PROGRAM AdsTcpUnit
VAR_OUTPUT
	bBusy : BOOL;
	err : BOOL;
	errid : UDINT;
END_VAR
VAR_OUTPUT
	areaSockets : ARRAY[1..6] OF POINTER TO AdsSocket; //only used for finding a socket by name
	subarea4Sockets : ARRAY[1..9] OF POINTER TO AdsSocket;
END_VAR
VAR	
	socket : REFERENCE TO AdsSocket;
	i : INT;
END_VAR

(*
this basic version of AdsTcp communication does not dynamically generate ADS messages into a queue to be polled cyclically
instead, modules must wait for the requested socket to finish sending its previous data before sending the next
*)

areaSockets[1] := ADR(AREA_1);
areaSockets[2] := ADR(AREA_2);
areaSockets[3] := ADR(AREA_3);
areaSockets[4] := ADR(AREA_4);
areaSockets[5] := ADR(AREA_5);
areaSockets[6] := ADR(AREA_6);

subarea4Sockets[1] := ADR(SUBAREA_4_1);
subarea4Sockets[2] := ADR(SUBAREA_4_2);
subarea4Sockets[3] := ADR(SUBAREA_4_3);
subarea4Sockets[4] := ADR(SUBAREA_4_4);
subarea4Sockets[5] := ADR(SUBAREA_4_5);
subarea4Sockets[6] := ADR(SUBAREA_4_6);
subarea4Sockets[7] := ADR(SUBAREA_4_7);
subarea4Sockets[8] := ADR(SUBAREA_4_8);
subarea4Sockets[9] := ADR(SUBAREA_4_9);

blocks();

METHOD PRIVATE blocks : BOOL
VAR_INPUT
END_VAR
(*
AREA_1(
	PrgName=> , 
	AmsNetId=> , 
	AmsPort=> , 
	receivingData=> , 
	sendingData=> , 
	readBusy=> , 
	readError=> , 
	readErrorId=> , 
	writeBusy=> , 
	writeError=> , 
	writeErrorId=> );
*)
(*
AREA_2(
	PrgName=> , 
	AmsNetId=> , 
	AmsPort=> , 
	receivingData=> , 
	sendingData=> , 
	readBusy=> , 
	readError=> , 
	readErrorId=> , 
	writeBusy=> , 
	writeError=> , 
	writeErrorId=> );
*)
(*
AREA_3(
	PrgName=> , 
	AmsNetId=> , 
	AmsPort=> , 
	receivingData=> , 
	sendingData=> , 
	readBusy=> , 
	readError=> , 
	readErrorId=> , 
	writeBusy=> , 
	writeError=> , 
	writeErrorId=> );
	
AREA_4(
	PrgName=> , 
	AmsNetId=> , 
	AmsPort=> , 
	receivingData=> , 
	sendingData=> , 
	readBusy=> , 
	readError=> , 
	readErrorId=> , 
	writeBusy=> , 
	writeError=> , 
	writeErrorId=> );
	
AREA_5(
	PrgName=> , 
	AmsNetId=> , 
	AmsPort=> , 
	receivingData=> , 
	sendingData=> , 
	readBusy=> , 
	readError=> , 
	readErrorId=> , 
	writeBusy=> , 
	writeError=> , 
	writeErrorId=> );
	
AREA_6(
	PrgName=> , 
	AmsNetId=> , 
	AmsPort=> , 
	receivingData=> , 
	sendingData=> , 
	readBusy=> , 
	readError=> , 
	readErrorId=> , 
	writeBusy=> , 
	writeError=> , 
	writeErrorId=> );
*)
END_METHOD

METHOD PRIVATE findSocket : REFERENCE TO AdsSocket
VAR_INPUT
	recipient : STRING;
END_VAR
FOR i:=1 TO numSockets BY 1 DO
	IF areaSockets[i] <> 0 AND_THEN areaSockets[i]^.PrgName = recipient THEN
		findSocket REF= areaSockets[i]^;
		RETURN;
	END_IF
END_FOR

FOR i:=1 TO numSubarea4Sockets BY 1 DO
	IF subarea4Sockets[i] <> 0 AND_THEN subarea4Sockets[i]^.PrgName = recipient THEN
		findSocket REF= areaSockets[i]^;
		RETURN;
	END_IF
END_FOR
END_METHOD

METHOD sendMessage : BOOL
VAR_INPUT
	recipient : STRING;
	data : REFERENCE TO AdsData;
END_VAR
VAR
	//socket : REFERENCE TO AdsSocket;
END_VAR
socket REF= findSocket(recipient := recipient);

IF __ISVALIDREF(socket) AND_THEN NOT socket.writeBusy THEN
	socket.send(data := data);
	sendMessage := TRUE;
END_IF
END_METHOD

END_PROGRAM

(* stored: Version 1.1.0.1, ProductVersion 3.1.4024.11
   POU AdsTcpUnit: Id {b856df85-9807-46f0-bd45-80629c76825c}, SpecialFunc None
   Method blocks: Id {6b41de23-37b5-4015-b6bc-69f9f2aa1377}
   Method findSocket: Id {9391686a-f9a5-427d-83ec-e84744570a4a}
   Method sendMessage: Id {1b1f9d8d-3fba-4fa0-976b-18f6d2359815} *)
